{attribute 'Tc2GvlVarNames'}
VAR_GLOBAL PERSISTENT
	gPrograms:ARRAY[1..MAX_NUMBER_OF_PROGRAMS] OF ST_PROGRAM;
	gCurrentProgram:ST_PROGRAM;
	giProgramNumber:INT;
END_VAR

(* stored: Version 1.1.0.1, ProductVersion 3.1.4024.10
   GVL PROGRAMS: Id {e89a6d2e-aa75-4ac0-b880-862caec8b34e} *)
